# EPICS autosave request: eigerApp/Db/eiger2_settings.req
file "eigerBase_settings.req", P=$(P), R=$(R)
$(P)$(R)Threshold1Enable
$(P)$(R)Threshold2Energy
$(P)$(R)Threshold2Enable
$(P)$(R)ThresholdDiffEnable
$(P)$(R)ExtGateMode
$(P)$(R)CountingMode
$(P)$(R)TriggerStartDelay
$(P)$(R)HVResetTime
